// TIA Portal V19 export
TYPE "C501_VAR_IF_HYK_TYPIC"
   STRUCT
      DEC { ExternalAccessible := 'False'; ExternalVisible := 'False'; ExternalWritable := 'False'} : Bool;   // De hydrantkast in de verkeerskoker is gesloten
      EXT_HW { ExternalAccessible := 'False'; ExternalVisible := 'False'; ExternalWritable := 'False'} : Bool;   // Sturings hardware (PLC) in storing
      STO { ExternalAccessible := 'False'; ExternalVisible := 'False'; ExternalWritable := 'False'} : Struct   // Opsomming van alle storingen
         A001 : Bool;   // Beveiliging aangesproken
         A002 : Bool;   // Temperatuur te laag
      END_STRUCT;
   END_STRUCT;
END_TYPE
